Fanuc TP program (LS listing): MON_OP20_ALM1.LS

/PROG  MON_OP20_ALM1
/ATTR
OWNER		= MNEDITOR;
COMMENT		= "MONITOR ALARM";
PROG_SIZE	= 271;
CREATE		= DATE 20-02-06  TIME 23:04:58;
MODIFIED	= DATE 20-02-06  TIME 23:04:58;
FILE_NAME	= MON_OP20;
VERSION		= 0;
LINE_COUNT	= 3;
MEMORY_SIZE	= 647;
PROTECT		= READ_WRITE;
TCD:  STACK_SIZE	= 0,
      TASK_PRIORITY	= 50,
      TIME_SLICE	= 0,
      BUSY_LAMP_OFF	= 0,
      ABORT_REQUEST	= 0,
      PAUSE_REQUEST	= 0;
DEFAULT_GROUP	= *,*,*,*,*;
CONTROL_CODE	= 00000000 00000000;
/APPL

AUTO_SINGULARITY_HEADER;
  ENABLE_SINGULARITY_AVOIDANCE   : TRUE;
/MN
   1:  CALL MACH_MSG(15) ;
   2:  UALM[5] ;
   3:  MONITOR MON_OP20_2 ;
/POS
/END
